// TIA Portal project "Calculator_webserver" (V17)

(* hardware
DEVICE "S71500/ET200MP station_9"  S7-1500 station
   slot 0: "Rail_0"  6ES7 590-1***0-0AA0
   slot 1: "PLC1"  CPU 1511-1 PN  6ES7 511-1AK01-0AB0  V2.0
      slot 3: "CPU display_1"  6ES7591-1AA00-0AA0
*)

// ===== PLC "PLC1"  CPU 1511-1 PN =====

VAR_GLOBAL   // PLC tag table "Default tag table"
   "NUMBER1" AT %MD100 : Real;
   "NUMBER2" AT %MD104 : Real;
   "OPERATION" AT %MB210 : Char;
   "ADD" AT %M108.0 : Bool;
   "RESULT" AT %MD109 : Real;
   "SUB" AT %M108.1 : Bool;
   "MUL" AT %M108.2 : Bool;
   "DIV" AT %M108.3 : Bool;
   "SQR" AT %M108.4 : Bool;
   "SQRT" AT %M108.5 : Bool;
END_VAR

DATA_BLOCK "ResultDB"   // DB1
{ S7_Optimized_Access := 'TRUE' }
VERSION : 0.1
   VAR
      NUMBER1_DISPLAY : Real;
      NUMBER2_DISPLAY : Real;
      OPERATION_DISPLAY : Char;
      RESULT_DISPLAY : Real;
   END_VAR
BEGIN
END_DATA_BLOCK

FUNCTION "Choose_operation" : Void   // FC1, SCL
{ S7_Optimized_Access := 'TRUE' }
VERSION : 0.1
   VAR_INPUT
      sign : Char;
   END_VAR
   VAR_OUTPUT
      add : Bool;
      sub : Bool;
      mul : Bool;
      sqr : Bool;
      sqrt : Bool;
      div : Bool;
   END_VAR
BEGIN
   #add := #sign = '+';
   #sub := #sign = '-';
   #mul := #sign = '*';
   #div := #sign = '/';
   #sqr := #sign = 's';
   #sqrt := #sign = 'p';
END_FUNCTION

FUNCTION "Copy_result" : Void   // FC2, SCL
{ S7_Optimized_Access := 'TRUE' }
VERSION : 0.1
   VAR_INPUT
      Num1 : Real;
      Num2 : Real;
      Res : Real;
      Operation : Char;
   END_VAR
   VAR_OUTPUT
      Num1_display : Real;
      Num2_display : Real;
      Res_display : Real;
      Operation_display : Char;
   END_VAR
BEGIN
   #Num1_display := #Num1;
   #Num2_display := #Num2;
   #Res_display := #Res;
   #Operation_display := #Operation;
END_FUNCTION

ORGANIZATION_BLOCK "Main"   // OB1, LAD, ProgramCycle
TITLE = "Main Program Sweep (Cycle)"
{ S7_Optimized_Access := 'TRUE' }
VERSION : 0.1
// //============================================================================
// // SIEMENS AG
// // (c)Copyright 2015 
// //-----------------------------------------------------------------------------
// // Library: ----
// // Tested with: TIA Portal V13 SP1
// // Engineering: TIA Portal V13 SP1
// // Restrictions: Main-OB
// // Requirements: PC with TIA-Portal and Browser, PLC (S7-1200 / S7-1500)
// // Functionality: WWW-function
// //-----------------------------------------------------------------------------
// // Change log table:
// // Version    Date           Expert in charge                                 Changes applied
// // 02.00.00 22.04.15    Siemens Industry Online Support   First released version
// //===========================================================================
// //============================================================================
// // SIEMENS AG
// // (c)Copyright 2015 All Rights Reserved
// //-----------------------------------------------------------------------------
// // Library: ----
// // Tested with: TIA Portal V13 SP1
// // Engineering: TIA Portal V13 SP1
// // Restrictions: Main-OB
// // Requirements: PC with TIA-Portal and Browser, PLC (S7-1200 / S7-1500)
// // Functionality: WWW-function
// //-----------------------------------------------------------------------------
// // Change log table:
// // Version    Date
// // 02.00.00 22.04.15 
// //===========================================================================
   VAR_INPUT
      Initial_Call : Bool;   // Initial call of this OB
      Remanence : Bool;   // =True, if remanent data are available
   END_VAR
   VAR_TEMP
      tempWwwRetVal : Int;
   END_VAR
   VAR_TEMP   // added for the SCL form of the ladder/FBD networks
      _w1 : Bool;
   END_VAR
BEGIN

REGION Network 1: WWW-function
   // initialize the webserver
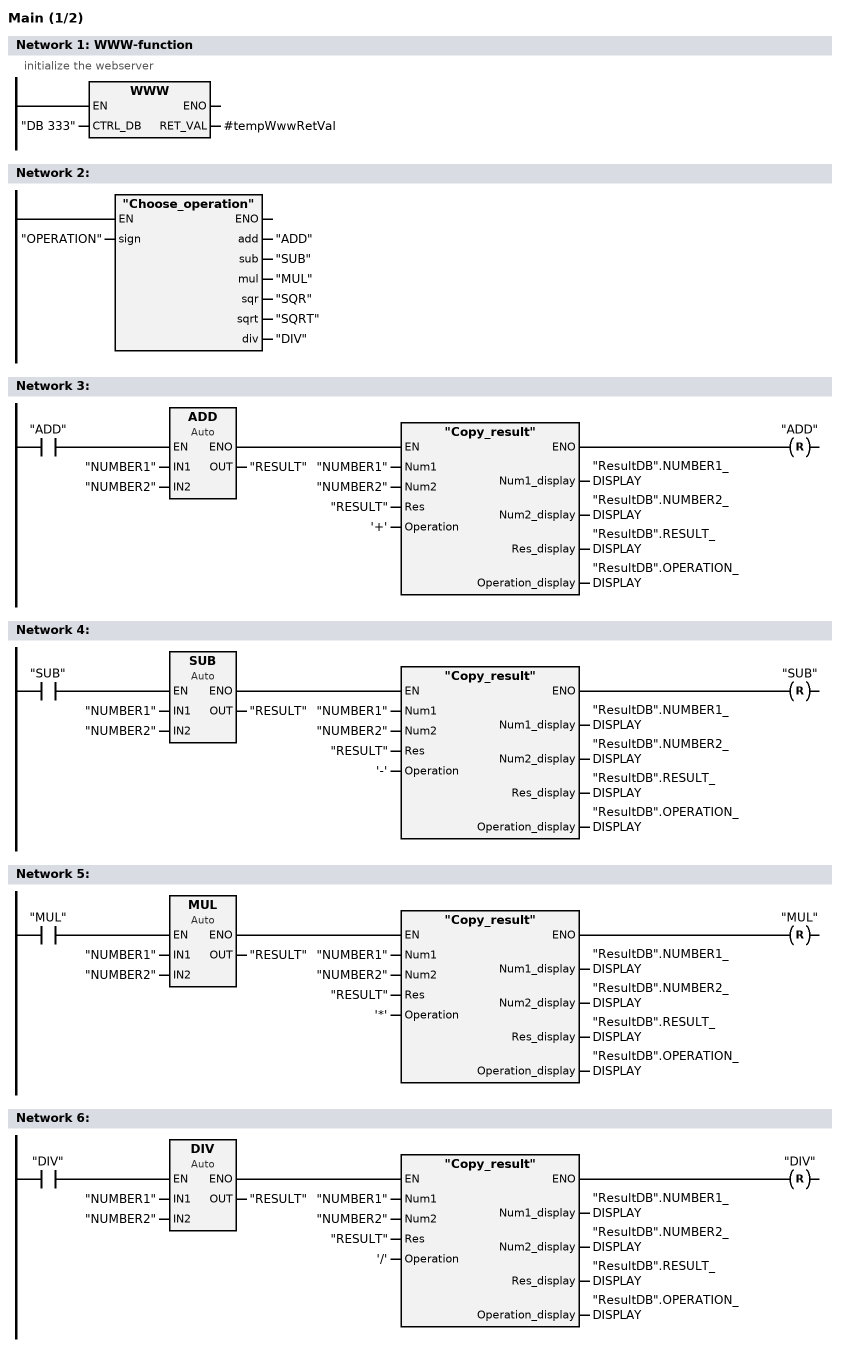
   #tempWwwRetVal := WWW(CTRL_DB := "DB 333");
END_REGION

REGION Network 2
   RUNG wire#powerrail
      "Choose_operation"(sign := "OPERATION", add => "ADD", sub => "SUB", mul => "MUL", sqr => "SQR", sqrt => "SQRT", div => "DIV")
   END_RUNG
   // the same network as SCL:
   "Choose_operation"(sign := "OPERATION",
                      add => "ADD",
                      sub => "SUB",
                      mul => "MUL",
                      sqr => "SQR",
                      sqrt => "SQRT",
                      div => "DIV");
END_REGION

REGION Network 3
   RUNG wire#powerrail
      Contact( "ADD" )
      Add(in1 := "NUMBER1", in2 := "NUMBER2", out => "RESULT")
      "Copy_result"(Num1 := "NUMBER1", Num2 := "NUMBER2", Res := "RESULT", Operation := '+', Num1_display => "ResultDB".NUMBER1_DISPLAY, Num2_display => "ResultDB".NUMBER2_DISPLAY, Res_display => "ResultDB".RESULT_DISPLAY, Operation_display => "ResultDB".OPERATION_DISPLAY)
      R_Coil( "ADD" )
   END_RUNG
   // the same network as SCL:
   IF "ADD" THEN "RESULT" := "NUMBER1" + "NUMBER2"; END_IF;
   "Copy_result"(EN := "ADD",
                 Num1 := "NUMBER1",
                 Num2 := "NUMBER2",
                 Res := "RESULT",
                 Operation := '+',
                 Num1_display => "ResultDB".NUMBER1_DISPLAY,
                 Num2_display => "ResultDB".NUMBER2_DISPLAY,
                 Res_display => "ResultDB".RESULT_DISPLAY,
                 Operation_display => "ResultDB".OPERATION_DISPLAY,
                 ENO => #_w1);
   IF #_w1 THEN "ADD" := FALSE; END_IF;
END_REGION

REGION Network 4
   RUNG wire#powerrail
      Contact( "SUB" )
      Sub(in1 := "NUMBER1", in2 := "NUMBER2", out => "RESULT")
      "Copy_result"(Num1 := "NUMBER1", Num2 := "NUMBER2", Res := "RESULT", Operation := '-', Num1_display => "ResultDB".NUMBER1_DISPLAY, Num2_display => "ResultDB".NUMBER2_DISPLAY, Res_display => "ResultDB".RESULT_DISPLAY, Operation_display => "ResultDB".OPERATION_DISPLAY)
      R_Coil( "SUB" )
   END_RUNG
   // the same network as SCL:
   IF "SUB" THEN "RESULT" := "NUMBER1" - "NUMBER2"; END_IF;
   "Copy_result"(EN := "SUB",
                 Num1 := "NUMBER1",
                 Num2 := "NUMBER2",
                 Res := "RESULT",
                 Operation := '-',
                 Num1_display => "ResultDB".NUMBER1_DISPLAY,
                 Num2_display => "ResultDB".NUMBER2_DISPLAY,
                 Res_display => "ResultDB".RESULT_DISPLAY,
                 Operation_display => "ResultDB".OPERATION_DISPLAY,
                 ENO => #_w1);
   IF #_w1 THEN "SUB" := FALSE; END_IF;
END_REGION

REGION Network 5
   RUNG wire#powerrail
      Contact( "MUL" )
      Mul(in1 := "NUMBER1", in2 := "NUMBER2", out => "RESULT")
      "Copy_result"(Num1 := "NUMBER1", Num2 := "NUMBER2", Res := "RESULT", Operation := '*', Num1_display => "ResultDB".NUMBER1_DISPLAY, Num2_display => "ResultDB".NUMBER2_DISPLAY, Res_display => "ResultDB".RESULT_DISPLAY, Operation_display => "ResultDB".OPERATION_DISPLAY)
      R_Coil( "MUL" )
   END_RUNG
   // the same network as SCL:
   IF "MUL" THEN "RESULT" := "NUMBER1" * "NUMBER2"; END_IF;
   "Copy_result"(EN := "MUL",
                 Num1 := "NUMBER1",
                 Num2 := "NUMBER2",
                 Res := "RESULT",
                 Operation := '*',
                 Num1_display => "ResultDB".NUMBER1_DISPLAY,
                 Num2_display => "ResultDB".NUMBER2_DISPLAY,
                 Res_display => "ResultDB".RESULT_DISPLAY,
                 Operation_display => "ResultDB".OPERATION_DISPLAY,
                 ENO => #_w1);
   IF #_w1 THEN "MUL" := FALSE; END_IF;
END_REGION

REGION Network 6
   RUNG wire#powerrail
      Contact( "DIV" )
      Div(in1 := "NUMBER1", in2 := "NUMBER2", out => "RESULT")
      "Copy_result"(Num1 := "NUMBER1", Num2 := "NUMBER2", Res := "RESULT", Operation := '/', Num1_display => "ResultDB".NUMBER1_DISPLAY, Num2_display => "ResultDB".NUMBER2_DISPLAY, Res_display => "ResultDB".RESULT_DISPLAY, Operation_display => "ResultDB".OPERATION_DISPLAY)
      R_Coil( "DIV" )
   END_RUNG
   // the same network as SCL:
   IF "DIV" THEN "RESULT" := "NUMBER1" / "NUMBER2"; END_IF;
   "Copy_result"(EN := "DIV",
                 Num1 := "NUMBER1",
                 Num2 := "NUMBER2",
                 Res := "RESULT",
                 Operation := '/',
                 Num1_display => "ResultDB".NUMBER1_DISPLAY,
                 Num2_display => "ResultDB".NUMBER2_DISPLAY,
                 Res_display => "ResultDB".RESULT_DISPLAY,
                 Operation_display => "ResultDB".OPERATION_DISPLAY,
                 ENO => #_w1);
   IF #_w1 THEN "DIV" := FALSE; END_IF;
END_REGION

REGION Network 7
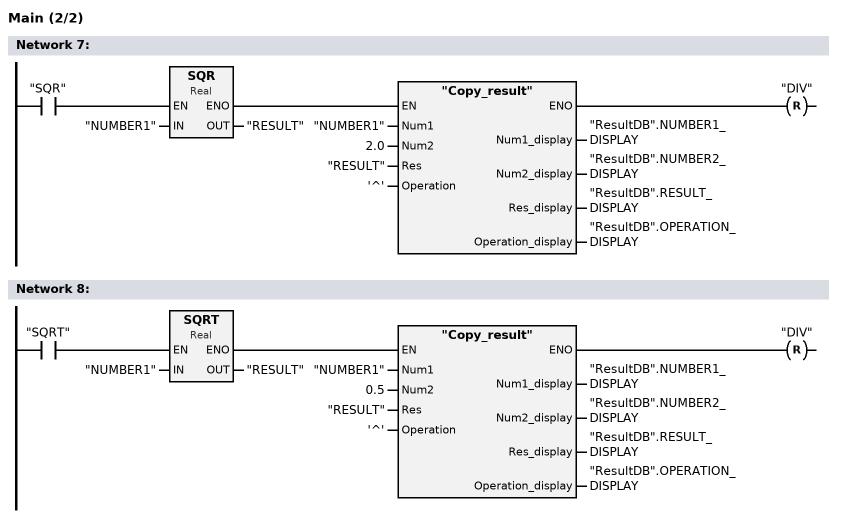
   IF "SQR" THEN "RESULT" := SQR("NUMBER1"); END_IF;
   "Copy_result"(EN := "SQR",
                 Num1 := "NUMBER1",
                 Num2 := 2.0,
                 Res := "RESULT",
                 Operation := '^',
                 Num1_display => "ResultDB".NUMBER1_DISPLAY,
                 Num2_display => "ResultDB".NUMBER2_DISPLAY,
                 Res_display => "ResultDB".RESULT_DISPLAY,
                 Operation_display => "ResultDB".OPERATION_DISPLAY,
                 ENO => #_w1);
   IF #_w1 THEN "DIV" := FALSE; END_IF;
END_REGION

REGION Network 8
   IF "SQRT" THEN "RESULT" := SQRT("NUMBER1"); END_IF;
   "Copy_result"(EN := "SQRT",
                 Num1 := "NUMBER1",
                 Num2 := 0.5,
                 Res := "RESULT",
                 Operation := '^',
                 Num1_display => "ResultDB".NUMBER1_DISPLAY,
                 Num2_display => "ResultDB".NUMBER2_DISPLAY,
                 Res_display => "ResultDB".RESULT_DISPLAY,
                 Operation_display => "ResultDB".OPERATION_DISPLAY,
                 ENO => #_w1);
   IF #_w1 THEN "DIV" := FALSE; END_IF;
END_REGION
END_ORGANIZATION_BLOCK

// ===== library types =====

// folder: Webserver

FUNCTION "WEB_Append_1BitToAsciiString" : Void   // FC1, SCL
TITLE = WEB_Append_1BitToAsciiString
{ S7_Optimized_Access := 'TRUE' }
AUTHOR : B.Geier
FAMILY : WebConv
// Convert a BOOL (1 Bit) to STRING
// '0' or '1'
   VAR_INPUT
      InBool : Bool;   // value as BOOL to convert into ASCII-String
   END_VAR
   VAR_IN_OUT
      AsciiString : String[254];   // ASCII String to append converted Value
   END_VAR
   VAR_TEMP
      tempChar : Char;   // temp CAHR to save ASCII value for ASCII String
   END_VAR
   VAR CONSTANT
      statTrue : Char := '1';
      statFalse : Char := '0';
   END_VAR
BEGIN
   //=============================================================================
   // Siemens
   // (c)Copyright (2015) All Rights Reserved
   //-----------------------------------------------------------------------------
   // Library: Simatic Webserver
   // Tested with: S7 1512SP v1.7
   // Engineering: TIA Portal (V13 SP1 UP5)
   // Restrictions: none
   // Requirements: 
   // Functionality: convert variables into Hex ASCII representation
   //-----------------------------------------------------------------------------
   // Change log table:
   // Version Date Expert in charge Changes applied
   // 00.00.01 29.10.2015 (Geier B.) First released LIB version, Styleguide
   //=============================================================================

   IF #InBool THEN // if TRUE
       #tempChar := #statTrue;
   ELSE // if FALSE
       #tempChar := #statFalse;
   END_IF;
   // copy TEMP Char to IN/OUT String
   #AsciiString := CONCAT(IN1 := #AsciiString, IN2 := #tempChar);
END_FUNCTION

FUNCTION "WEB_Append_8BitToAsciiString" : Void   // FC2, SCL
TITLE = WEB_Append_8BitToAsciiString
{ S7_Optimized_Access := 'TRUE' }
AUTHOR : B.Geier
FAMILY : WebConv
// Convert a BYTE (8 Bit / 1 Byte / 2 nibble) to STRING of max 2 characters
// In := BYTE to convert, starting by LSB of BYTE
   VAR_INPUT
      InByte : Byte;   // value as BYTE to convert into ASCII-String
   END_VAR
   VAR_IN_OUT
      AsciiString : String[254];   // ASCII String to append converted Value
   END_VAR
   VAR_TEMP
      tempIndex : SInt;   // how many nibbles to convert
      tempUSInt : USInt;   // temp nibble storage to convert in to ASCII Char
      tempString : String[2];   // temp String to build ASCII String from variable
   END_VAR
   VAR CONSTANT
      statCount : SInt := 2;   // how many nibbles to convert
      statString : String := '00';   // start value for string
      statMask : Byte := 16#0F;   // mask for nibbles
   END_VAR
BEGIN
   //=============================================================================
   // Siemens
   // (c)Copyright (2015) All Rights Reserved
   //-----------------------------------------------------------------------------
   // Library: Simatic Webserver
   // Tested with: S7 1512SP v1.7
   // Engineering: TIA Portal (V13 SP1 UP5)
   // Restrictions: none
   // Requirements: 
   // Functionality: convert variables into Hex ASCII representation
   //-----------------------------------------------------------------------------
   // Change log table:
   // Version Date Expert in charge Changes applied
   // 00.00.01 29.10.2015 (Geier B.) First released LIB version, Styleguide
   //=============================================================================

   // Loop trough input variable and calculate characters
   #tempIndex := #statCount;
   #tempString := #statString;
   WHILE #tempIndex > 0 DO
       #tempUSInt := BYTE_TO_USINT(#InByte AND #statMask); // get last nibble from BYTE to convert into char

     IF #tempUSInt < 10 THEN    // if smaller add '0'
       #tempUSInt := #tempUSInt + 48;
     ELSE                    // if greater add 'A'-10
       #tempUSInt := #tempUSInt + 55;
     END_IF;

     #tempString[#tempIndex] := USINT_TO_CHAR(#tempUSInt); // add char to temp string
     #InByte := SHR(IN := #InByte, N := 4); // shift to next nibble
     #tempIndex := #tempIndex - 1; // decrement index
   END_WHILE;
   // copy TEMP String to IN/OUT String
   #AsciiString := CONCAT(IN1 := #AsciiString, IN2 := #tempString);
END_FUNCTION

FUNCTION "WEB_Append_16BitToAsciiString" : Void   // FC5, SCL
TITLE = WEB_Append_16BitToAsciiString
{ S7_Optimized_Access := 'TRUE' }
AUTHOR : B.Geier
FAMILY : WebConv
// Convert a WORD (16 Bit / 2 Byte / 4 nibble) to STRING of max 4 characters
// In := WORD to convert, starting by LSB of WORD
   VAR_INPUT
      InWord : Word;   // value as WORD to convert into ASCII-String
   END_VAR
   VAR_IN_OUT
      AsciiString : String[254];   // ASCII String to append converted Value
   END_VAR
   VAR_TEMP
      tempIndex : SInt;   // how many nibbles to convert
      tempUSInt : USInt;   // temp nibble storage to convert in to ASCII Char
      tempString : String[4];   // temp String to build ASCII String from variable
   END_VAR
   VAR CONSTANT
      statCount : SInt := 4;   // how many nibbles to convert
      statString : String := '0000';   // start value for string
      statMask : Byte := 16#0F;   // mask for nibbles
   END_VAR
BEGIN
   //=============================================================================
   // Siemens
   // (c)Copyright (2015) All Rights Reserved
   //-----------------------------------------------------------------------------
   // Library: Simatic Webserver
   // Tested with: S7 1512SP v1.7
   // Engineering: TIA Portal (V13 SP1 UP5)
   // Restrictions: none
   // Requirements: 
   // Functionality: convert variables into Hex ASCII representation
   //-----------------------------------------------------------------------------
   // Change log table:
   // Version Date Expert in charge Changes applied
   // 00.00.01 29.10.2015 (Geier B.) First released LIB version, Styleguide
   //=============================================================================

   // Loop trough input variable and calculate characters
   #tempIndex := #statCount;
   #tempString := #statString;
   WHILE #tempIndex > 0 DO
       #tempUSInt := WORD_TO_USINT(#InWord AND #statMask); // get last nibble from WORD to convert into char

       IF #tempUSInt < 10 THEN    // if smaller add '0'
          #tempUSInt := #tempUSInt + 48;
   ELSE                    // if greater add 'A'-10
       #tempUSInt := #tempUSInt + 55;
     END_IF;

     #tempString[#tempIndex] := USINT_TO_CHAR(#tempUSInt); // add char to temp string
     #InWord := SHR(IN := #InWord, N := 4); // shift to next nibble
     #tempIndex := #tempIndex - 1; // decrement index
   END_WHILE;
   // copy TEMP String to IN/OUT String
   #AsciiString := CONCAT(IN1 := #AsciiString, IN2 := #tempString);
END_FUNCTION

FUNCTION "WEB_Append_32BitToAsciiString" : Void   // FC6, SCL
TITLE = WEB_Append_32BitToAsciiString
{ S7_Optimized_Access := 'TRUE' }
AUTHOR : B.Geier
FAMILY : WebConv
// Convert a DWORD (32Bit / 4 Byte / 8 nibble) to STRING of max 8 characters
// In := DWORD to convert, starting by LSB of DWORD
   VAR_INPUT
      InDWord : DWord;   // value as DWORD to convert into ASCII-String
   END_VAR
   VAR_IN_OUT
      AsciiString : String[254];   // ASCII String to append converted Value
   END_VAR
   VAR_TEMP
      tempIndex : SInt;   // how many nibbles to convert
      tempUSInt : USInt;   // temp nibble storage to convert in to ASCII Char
      tempString : String[8];   // temp String to build ASCII String from variable
   END_VAR
   VAR CONSTANT
      statCount : SInt := 8;   // how many nibbles to convert
      statString : String := '00000000';   // start value for string
      statMask : Byte := 16#0F;   // mask for nibbles
   END_VAR
BEGIN
   //=============================================================================
   // Siemens
   // (c)Copyright (2015) All Rights Reserved
   //-----------------------------------------------------------------------------
   // Library: Simatic Webserver
   // Tested with: S7 1512SP v1.7
   // Engineering: TIA Portal (V13 SP1 UP5)
   // Restrictions: none
   // Requirements: 
   // Functionality: convert variables into Hex ASCII representation
   //-----------------------------------------------------------------------------
   // Change log table:
   // Version Date Expert in charge Changes applied
   // 00.00.01 29.10.2015 (Geier B.) First released LIB version, Styleguide
   //=============================================================================

   // Loop trough input variable and calculate characters
   #tempIndex := #statCount;
   #tempString := #statString;
   WHILE #tempIndex > 0 DO
       #tempUSInt := DWORD_TO_USINT(#InDWord AND #statMask); // get last nibble from DWORD to convert into char

       IF #tempUSInt < 10 THEN    // if smaller add '0'
       #tempUSInt := #tempUSInt + 48;
   ELSE                    // if greater add 'A'-10
       #tempUSInt := #tempUSInt + 55;
     END_IF;

     #tempString[#tempIndex] := USINT_TO_CHAR(#tempUSInt); // add char to temp string
     #InDWord := SHR(IN := #InDWord, N := 4); // shift to next nibble
     #tempIndex := #tempIndex - 1; // decrement index
   END_WHILE;
   // copy TEMP String to IN/OUT String
   #AsciiString := CONCAT(IN1 := #AsciiString, IN2 := #tempString);
END_FUNCTION